(* Schneider Machine Expert - Basic project es1_2pompe_1max_2soglie_alternanza_minor_numero_ore, file version 3.0.0.0 *)
(* ProjectInformations: Name=New project *)

HARDWARE
  Cpu 0: TM221C40R
  EthernetConfiguration: NetworkName=M221, IpAllocationMode=FixedAddress, IpAddress=0.0.0.0, SubnetMask=0.0.0.0
  SerialLineConfiguration: Baud=Baud19200, Parity=ParityEven, DataBits=DataBits8, StopBits=StopBits1, PhysicalMedium=PhysicalMediumRs485, TransmissionMode=TransmissionModeModbusRtu, SlaveId=1, Addressing=SlaveAddressing
  MastTask: UsePeriodScanMode=false, PeriodScan=100
  FastTask: Period=255
  CpuBehavior: StartingMode=StartAsPreviousState, AutoSaveRamOnEeprom=true, WatchdogPeriod=250

SYMBOLS  (address, symbol, comment, settings)
  %M0       P1_USABILE
  %M1       P2_USABILE
  %M2       P1_SUPERATO_NUMERO_SEC_LAVORATI
  %M3       P2_SUPERATO_NUMERO_SEC_LAVORATI
  %S6       SB_TB1S  "Time base of 1 s generated by an internal clock"
  %MW0      PROSSIMA_POMPA_CANDIDATA
  %TM0      TIMER_POMPA_1  [Preset=10, Base=OneSecond, IsRetentive=true, IsDynamicPreset=true]
  %C0       CONTATORE_P1_SECONDI_LAVORATI  [Preset=0]
  %C1       CONTATORE_P2_SECONDI_LAVORATI  [Preset=0]
  %I0.0     P1_AUTO
  %I0.1     P1_MOTO
  %I0.2     P1_ANOMALIA
  %I0.3     P2_AUTO
  %I0.4     P2_MOTO
  %I0.5     P2_ANOMALIA
  %I0.6     LVL_MIN
  %I0.7     LVL_MAX
  %Q0.0     P1_CMD
  %Q0.1     P2_CMD
  %IW0.0    NUMERO_MIN_PRESET  [Type=Type_0_10V, Scope=Scope_Normal, Minimum=0, Maximum=1000]

POU New POU
  (* SectionNumber=1 *)

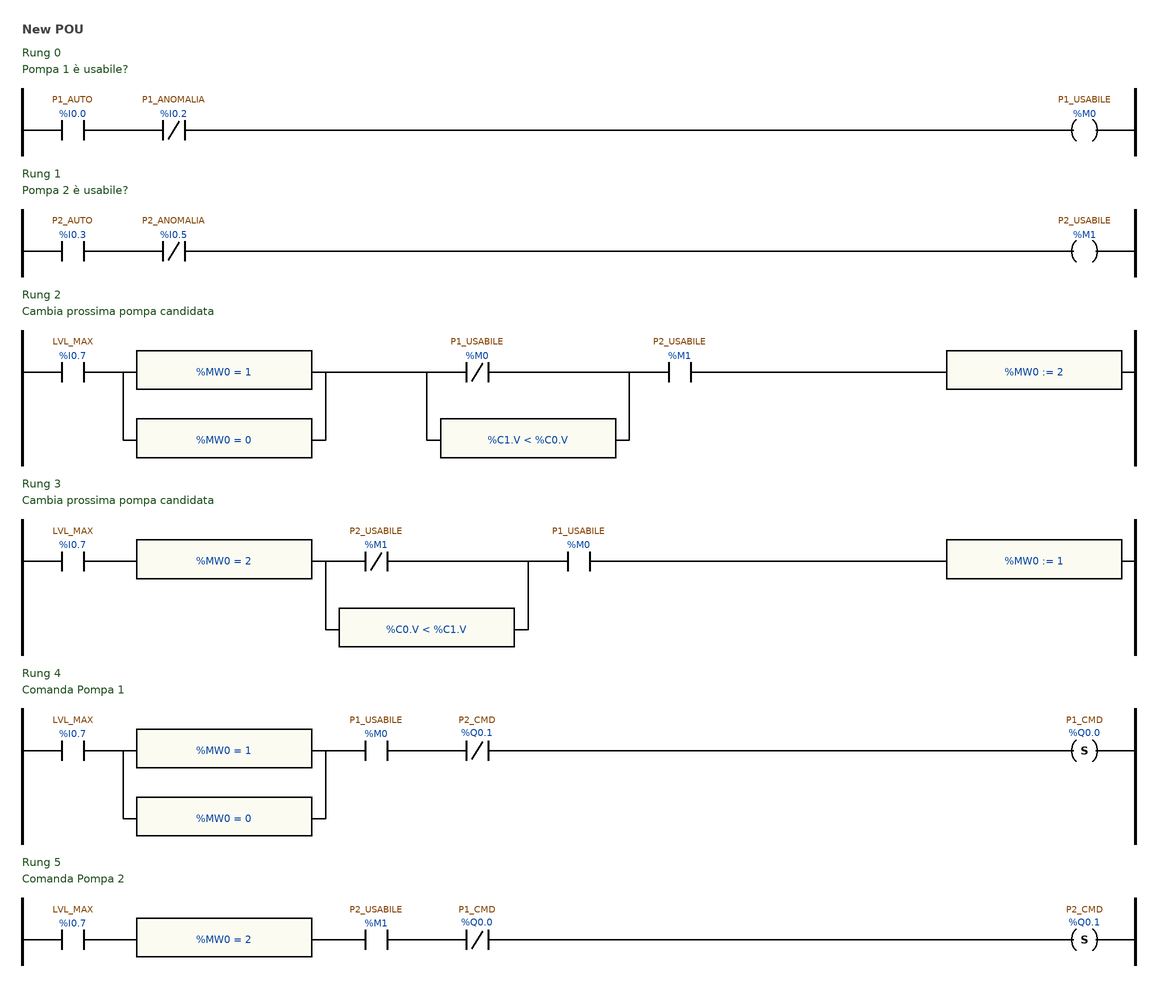

// Rung 0
// Pompa 1 è usabile?
  LD %I0.0                (* P1_AUTO *)
  ANDN %I0.2              (* P1_ANOMALIA *)
  ST %M0                  (* P1_USABILE *)
  // as ST:
  //   P1_USABILE := P1_AUTO AND NOT P1_ANOMALIA;

// Rung 1
// Pompa 2 è usabile?
  LD %I0.3                (* P2_AUTO *)
  ANDN %I0.5              (* P2_ANOMALIA *)
  ST %M1                  (* P2_USABILE *)
  // as ST:
  //   P2_USABILE := P2_AUTO AND NOT P2_ANOMALIA;

// Rung 2
// Cambia prossima pompa candidata
  LD %I0.7                (* LVL_MAX *)
  AND( [ %MW0 = 1 ]       (* PROSSIMA_POMPA_CANDIDATA *)
  OR [ %MW0 = 0 ]         (* PROSSIMA_POMPA_CANDIDATA *)
  )
  AND(N %M0               (* P1_USABILE *)
  OR [ %C1.V < %C0.V ]    (* CONTATORE_P2_SECONDI_LAVORATI, CONTATORE_P1_SECONDI_LAVORATI *)
  )
  AND %M1                 (* P2_USABILE *)
  [ %MW0 := 2 ]           (* PROSSIMA_POMPA_CANDIDATA *)
  // as ST:
  //   IF LVL_MAX AND (PROSSIMA_POMPA_CANDIDATA = 1 OR PROSSIMA_POMPA_CANDIDATA = 0) AND (NOT P1_USABILE OR CONTATORE_P2_SECONDI_LAVORATI.V < CONTATORE_P1_SECONDI_LAVORATI.V) AND P2_USABILE THEN PROSSIMA_POMPA_CANDIDATA := 2; END_IF;

// Rung 3
// Cambia prossima pompa candidata
  LD %I0.7                (* LVL_MAX *)
  AND [ %MW0 = 2 ]        (* PROSSIMA_POMPA_CANDIDATA *)
  AND(N %M1               (* P2_USABILE *)
  OR [ %C0.V < %C1.V ]    (* CONTATORE_P1_SECONDI_LAVORATI, CONTATORE_P2_SECONDI_LAVORATI *)
  )
  AND %M0                 (* P1_USABILE *)
  [ %MW0 := 1 ]           (* PROSSIMA_POMPA_CANDIDATA *)
  // as ST:
  //   IF LVL_MAX AND PROSSIMA_POMPA_CANDIDATA = 2 AND (NOT P2_USABILE OR CONTATORE_P1_SECONDI_LAVORATI.V < CONTATORE_P2_SECONDI_LAVORATI.V) AND P1_USABILE THEN PROSSIMA_POMPA_CANDIDATA := 1; END_IF;

// Rung 4
// Comanda Pompa 1
  LD %I0.7                (* LVL_MAX *)
  AND( [ %MW0 = 1 ]       (* PROSSIMA_POMPA_CANDIDATA *)
  OR [ %MW0 = 0 ]         (* PROSSIMA_POMPA_CANDIDATA *)
  )
  AND %M0                 (* P1_USABILE *)
  ANDN %Q0.1              (* P2_CMD *)
  S %Q0.0                 (* P1_CMD *)
  // as ST:
  //   IF LVL_MAX AND (PROSSIMA_POMPA_CANDIDATA = 1 OR PROSSIMA_POMPA_CANDIDATA = 0) AND P1_USABILE AND NOT P2_CMD THEN P1_CMD := TRUE; END_IF;

// Rung 5
// Comanda Pompa 2
  LD %I0.7                (* LVL_MAX *)
  AND [ %MW0 = 2 ]        (* PROSSIMA_POMPA_CANDIDATA *)
  AND %M1                 (* P2_USABILE *)
  ANDN %Q0.0              (* P1_CMD *)
  S %Q0.1                 (* P2_CMD *)
  // as ST:
  //   IF LVL_MAX AND PROSSIMA_POMPA_CANDIDATA = 2 AND P2_USABILE AND NOT P1_CMD THEN P2_CMD := TRUE; END_IF;

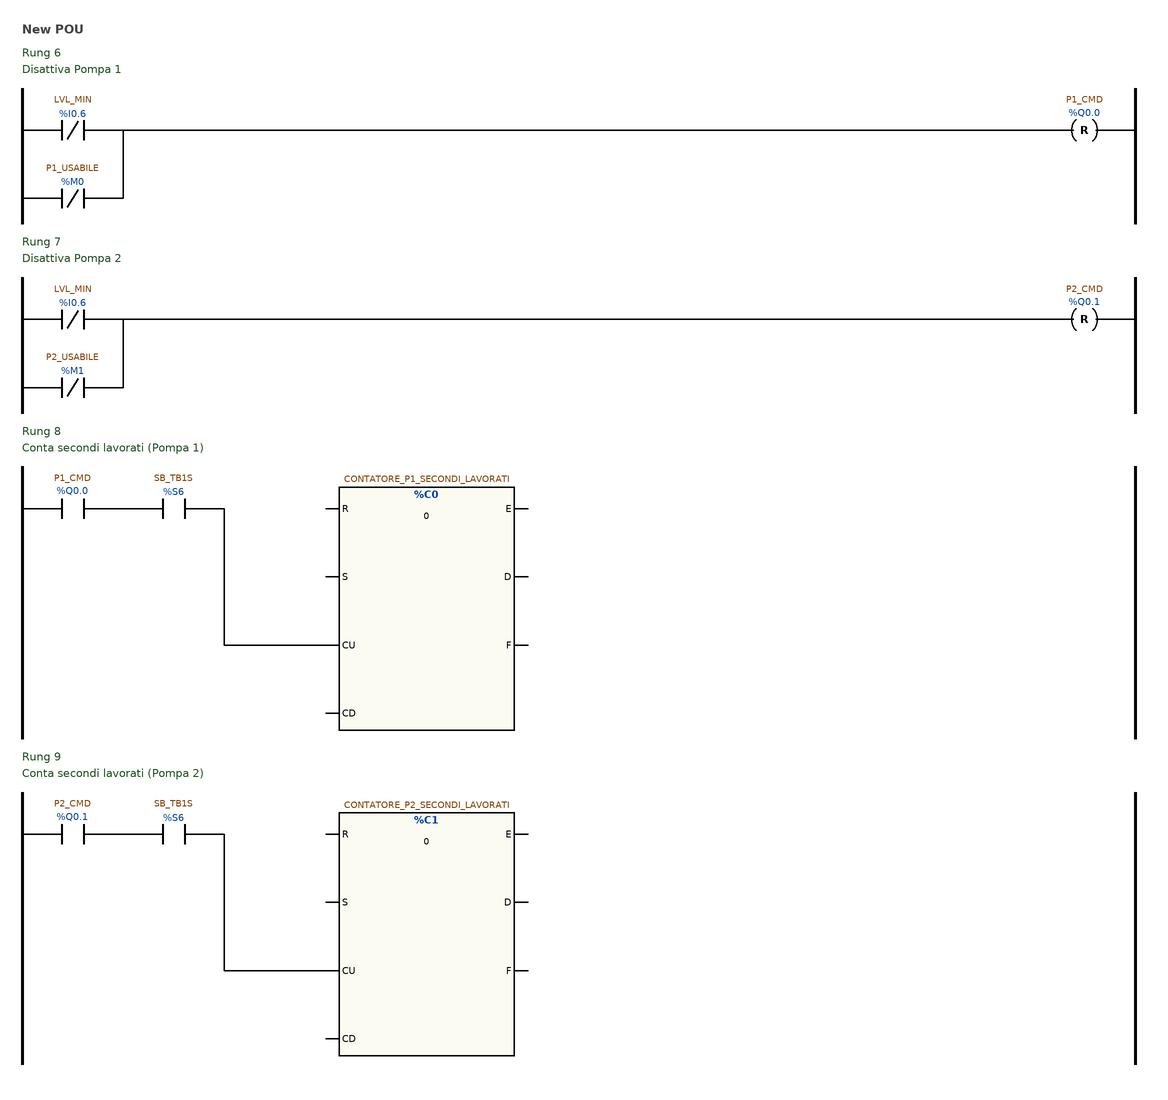

// Rung 6
// Disattiva Pompa 1
  LDN %I0.6               (* LVL_MIN *)
  ORN %M0                 (* P1_USABILE *)
  R %Q0.0                 (* P1_CMD *)
  // as ST:
  //   IF NOT LVL_MIN OR NOT P1_USABILE THEN P1_CMD := FALSE; END_IF;

// Rung 7
// Disattiva Pompa 2
  LDN %I0.6               (* LVL_MIN *)
  ORN %M1                 (* P2_USABILE *)
  R %Q0.1                 (* P2_CMD *)
  // as ST:
  //   IF NOT LVL_MIN OR NOT P2_USABILE THEN P2_CMD := FALSE; END_IF;

// Rung 8
// Conta secondi lavorati (Pompa 1)
  BLK %C0                 (* CONTATORE_P1_SECONDI_LAVORATI *)
  LD %Q0.0                (* P1_CMD *)
  AND %S6                 (* SB_TB1S *)
  CU
  END_BLK
  // as ST:
  //   CONTATORE_P1_SECONDI_LAVORATI(CU := P1_CMD AND SB_TB1S);

// Rung 9
// Conta secondi lavorati (Pompa 2)
  BLK %C1                 (* CONTATORE_P2_SECONDI_LAVORATI *)
  LD %Q0.1                (* P2_CMD *)
  AND %S6                 (* SB_TB1S *)
  CU
  END_BLK
  // as ST:
  //   CONTATORE_P2_SECONDI_LAVORATI(CU := P2_CMD AND SB_TB1S);
